(* PLC project Programme MGS_2-07_refactorJOY.project, CODESYS CODESYS V3.5 SP19 Patch 1 *)
(* stored: creationDateTime 2026-06-29T23:37:41.0776378, modificationDateTime 2026-06-29T22:49:33.424 *)

FUNCTION_BLOCK FB_Encoder_Scale
  VAR_INPUT
    CurrentRawPos : UDINT;  (* Valeur brute synchrone (%ID2) *)
    OffsetValueB : REAL;  (* Le "b" de l'équation (décalage en mètres) *)
    EnableTeach : BOOL;  (* Active le mode calibration *)
    StartTeachPos : UDINT;  (* Capture de la position brute au point A *)
    EndTeachPos : UDINT;  (* Capture de la position brute au point B *)
    RealDistMeters : REAL;  (* Distance réelle mesurée au mètre ruban entre A et B *)
  END_VAR
  VAR_IN_OUT
    PulsePerMeter : REAL;  (* Le "a" de l'équation (Pulsations / mètre) *)
  END_VAR
  VAR_OUTPUT
    PositionMeters : REAL;  (* La sortie finale f(x) = ax + b *)
  END_VAR
  VAR
    DeltaPulses : REAL;
  END_VAR

            // 1. Mode Teach : Calcul automatique du coefficient de mise à l'échelle (a)
IF EnableTeach AND RealDistMeters > 0.001 THEN
    DeltaPulses := UDINT_TO_REAL(EndTeachPos) - UDINT_TO_REAL(StartTeachPos);
    IF ABS(DeltaPulses) > 0.0 THEN
        // Calcul du ratio : impulsions par mètre
        PulsePerMeter := ABS(DeltaPulses) / RealDistMeters;
    END_IF
END_IF

// 2. Application de la formule affine y = ax + b
// Sécurité : évite la division par zéro si le ratio n'est pas configuré
IF PulsePerMeter > 0.001 THEN
    PositionMeters := (UDINT_TO_REAL(CurrentRawPos) / PulsePerMeter) + OffsetValueB;
ELSE
    PositionMeters := 0.0;
END_IF
          
END_FUNCTION_BLOCK
